FUNCTION_BLOCK ACVariobatch EXTENDS ACComponent IMPLEMENTS IACVariobatch
VAR_INPUT
END_VAR
VAR_OUTPUT
	// Metadata about Memory-Structure, Index in Array represents Instance-ID
	_Metadata : ARRAY [1..GCL.cMetaObjMAX] OF ACRMemoryMetaObj;
	// Copy of Memory
	_Memory : ARRAY [0..GCL.cMemorySizeMAX] OF BYTE;
	_MemorySizeUsed : UDINT;

	// Property-Changed-Notifications
	_EventsByte : ACRMemoryByteEvents;
	_EventsUInt : ACRMemoryUIntEvents;
	_EventsInt : ACRMemoryIntEvents;
	_EventsUDInt : ACRMemoryUDIntEvents;
	_EventsDInt : ACRMemoryDIntEvents;
	_EventsReal : ACRMemoryRealEvents;
	_EventsLReal : ACRMemoryLRealEvents;
	_EventsString : ACRMemoryStringEvents;
	_EventsTime : ACRMemoryTimeEvents;
	_EventsDT : ACRMemoryDTEvents;
	_EventCycleInfo : ACREventCycleInfo; 
	_MemPropEventCycle : ARRAY [1..GCL.cMetaObjMAX, 1..GCL.cMetaPropMAX] OF ACREventCycleProp;
	
	_InSimulation : BOOL;
	END_VAR
VAR
END_VAR

METHOD PUBLIC FB_postinit
VAR_INPUT
		root : IACVariobatch;
END_VAR
ResetMemory();
SUPER^.FB_postinit(root);
END_METHOD

PROPERTY InSimulation : BOOL
GET
InSimulation := _InSimulation;
END_GET
END_PROPERTY

METHOD OnObjectMetaBuilded
VAR_INPUT
	iObject : IACObject;
END_VAR
VAR
	instanceID : UDINT;
	memorySizeToObject : UDINT;
	i : UINT;
	offset : WORD;
END_VAR
instanceID := iObject.InstanceID;
offset := 0;

IF instanceID > 1 THEN
	_Metadata[instanceID]._OffsetInMemory := _Metadata[instanceID-1]._MetaPropSize + _Metadata[instanceID-1]._OffsetInMemory;
END_IF

IF iObject.MaxPropertyID >= 1 THEN
	FOR i:=1 TO iObject.MaxPropertyID BY 1
	  DO
		IF (_Metadata[instanceID]._MetaProp[i]._Length > 0) THEN
			_Metadata[instanceID]._MetaProp[i]._Offset := offset;
			offset := offset + _Metadata[instanceID]._MetaProp[i]._Length;
		//ELSE
			//EXIT;
		END_IF
	END_FOR;
END_IF

_Metadata[instanceID]._MaxPropertyID := iObject.MaxPropertyID;
_Metadata[instanceID]._MetaPropSize := offset;
memorySizeToObject := _Metadata[instanceID]._OffsetInMemory + offset;

IF _MemorySizeUsed < memorySizeToObject THEN
	_MemorySizeUsed := memorySizeToObject;
END_IF
END_METHOD

METHOD PUBLIC OnPropertyChangedBool
VAR_INPUT
	object : IACObject;
	propertyID : UINT;
	value : BOOL;
END_VAR
VAR
	instanceID : UDINT;
	memAdr : UDINT;
	eventIndex : DINT;
END_VAR
instanceID := object.InstanceID;
// 1. Copy to memory
memAdr := _Metadata[instanceID]._OffsetInMemory + _Metadata[instanceID]._MetaProp[propertyID]._Offset;
IF value THEN
	_Memory[memAdr] := 1;
ELSE
	_Memory[memAdr] := 0;
END_IF

// 2. Add to Eventlist
IF _EventCycleInfo._MemReadCycle = _EventCycleInfo._MemWriteCycle THEN
	IF _EventCycleInfo._MemWriteCycle > GCL.cMemoryEventCycleMAX THEN
		_EventCycleInfo._MemWriteCycle := 0;
	END_IF
	_EventCycleInfo._MemWriteCycle := _EventCycleInfo._MemWriteCycle + 1;
END_IF

IF _MemPropEventCycle[instanceID, propertyID]._MemWriteCycle = _EventCycleInfo._MemWriteCycle THEN
	eventIndex := _MemPropEventCycle[instanceID, propertyID]._MemEventPos;
ELSE
	eventIndex := _EventCycleInfo._NextByteEventIndex;
	IF eventIndex < 0 OR eventIndex > GCL.cMemoryEventsMAX THEN
		eventIndex := 0;
	END_IF	
	_MemPropEventCycle[instanceID, propertyID]._MemEventPos := eventIndex;
	_MemPropEventCycle[instanceID, propertyID]._MemWriteCycle := _EventCycleInfo._MemWriteCycle;
	_EventCycleInfo._NextByteEventIndex := eventIndex + 1;
END_IF

_EventsByte._Values[eventIndex]._InstanceID := instanceID;
_EventsByte._Values[eventIndex]._PropertyID := propertyID;
_EventsByte._Values[eventIndex]._Value := _Memory[memAdr];
END_METHOD

METHOD PUBLIC OnPropertyChangedByte
VAR_INPUT
	object : IACObject;
	propertyID : UINT;
	value : BYTE;
END_VAR
VAR
	instanceID : UDINT;
	memAdr : UDINT;
	eventIndex : DINT;
END_VAR
instanceID := object.InstanceID;

// 1. Copy to memory
memAdr := _Metadata[instanceID]._OffsetInMemory + _Metadata[instanceID]._MetaProp[propertyID]._Offset;
_Memory[memAdr] := value;

// 2. Add to Eventlist
IF _EventCycleInfo._MemReadCycle = _EventCycleInfo._MemWriteCycle THEN
	IF _EventCycleInfo._MemWriteCycle > GCL.cMemoryEventCycleMAX THEN
		_EventCycleInfo._MemWriteCycle := 0;
	END_IF
	_EventCycleInfo._MemWriteCycle := _EventCycleInfo._MemWriteCycle + 1;
END_IF

IF _MemPropEventCycle[instanceID, propertyID]._MemWriteCycle = _EventCycleInfo._MemWriteCycle THEN
	eventIndex := _MemPropEventCycle[instanceID, propertyID]._MemEventPos;
ELSE
	eventIndex := _EventCycleInfo._NextByteEventIndex;
	IF eventIndex < 0 OR eventIndex > GCL.cMemoryEventsMAX THEN
		eventIndex := 0;
	END_IF	
	_MemPropEventCycle[instanceID, propertyID]._MemEventPos := eventIndex;
	_MemPropEventCycle[instanceID, propertyID]._MemWriteCycle := _EventCycleInfo._MemWriteCycle;
	_EventCycleInfo._NextByteEventIndex := eventIndex + 1;
END_IF

_EventsByte._Values[eventIndex]._InstanceID := instanceID;
_EventsByte._Values[eventIndex]._PropertyID := propertyID;
_EventsByte._Values[eventIndex]._Value := value;
END_METHOD

METHOD PUBLIC OnPropertyChangedDInt
VAR_INPUT
	object : IACObject;
	propertyID : UINT;
	value : DINT;
END_VAR
VAR
	instanceID : UDINT;
	memAdr : UDINT;
	eventIndex : DINT;
END_VAR
instanceID := object.InstanceID;

// 1. Copy to memory
memAdr := _Metadata[instanceID]._OffsetInMemory + _Metadata[instanceID]._MetaProp[propertyID]._Offset;
MEMCPY(ADR(_Memory[memAdr]), ADR(value), GCL.cSizeDINT);

// 2. Add to Eventlist
IF _EventCycleInfo._MemReadCycle = _EventCycleInfo._MemWriteCycle THEN
	IF _EventCycleInfo._MemWriteCycle > GCL.cMemoryEventCycleMAX THEN
		_EventCycleInfo._MemWriteCycle := 0;
	END_IF
	_EventCycleInfo._MemWriteCycle := _EventCycleInfo._MemWriteCycle + 1;
END_IF

IF _MemPropEventCycle[instanceID, propertyID]._MemWriteCycle = _EventCycleInfo._MemWriteCycle THEN
	eventIndex := _MemPropEventCycle[instanceID, propertyID]._MemEventPos;
ELSE
	eventIndex := _EventCycleInfo._NextDIntEventIndex;
	IF eventIndex < 0 OR eventIndex > GCL.cMemoryEventsMAX THEN
		eventIndex := 0;
	END_IF	
	_MemPropEventCycle[instanceID, propertyID]._MemEventPos := eventIndex;
	_MemPropEventCycle[instanceID, propertyID]._MemWriteCycle := _EventCycleInfo._MemWriteCycle;
	_EventCycleInfo._NextDIntEventIndex := eventIndex + 1;
END_IF

_EventsDInt._Values[eventIndex]._InstanceID := instanceID;
_EventsDInt._Values[eventIndex]._PropertyID := propertyID;
_EventsDInt._Values[eventIndex]._Value := value;
END_METHOD

METHOD PUBLIC OnPropertyChangedDT
VAR_INPUT
	object : IACObject;
	propertyID : UINT;
	value : DATE_AND_TIME;
END_VAR
VAR
	instanceID : UDINT;
	memAdr : UDINT;
	eventIndex : DINT;
END_VAR
instanceID := object.InstanceID;

// 1. Copy to memory
memAdr := _Metadata[instanceID]._OffsetInMemory + _Metadata[instanceID]._MetaProp[propertyID]._Offset;
MEMCPY(ADR(_Memory[memAdr]), ADR(value), GCL.cSizeDT);

// 2. Add to Eventlist
IF _EventCycleInfo._MemReadCycle = _EventCycleInfo._MemWriteCycle THEN
	IF _EventCycleInfo._MemWriteCycle > GCL.cMemoryEventCycleMAX THEN
		_EventCycleInfo._MemWriteCycle := 0;
	END_IF
	_EventCycleInfo._MemWriteCycle := _EventCycleInfo._MemWriteCycle + 1;
END_IF

IF _MemPropEventCycle[instanceID, propertyID]._MemWriteCycle = _EventCycleInfo._MemWriteCycle THEN
	eventIndex := _MemPropEventCycle[instanceID, propertyID]._MemEventPos;
ELSE
	eventIndex := _EventCycleInfo._NextDTEventIndex;
	IF eventIndex < 0 OR eventIndex > GCL.cMemoryEventsMidMAX THEN
		eventIndex := 0;
	END_IF	
	_MemPropEventCycle[instanceID, propertyID]._MemEventPos := eventIndex;
	_MemPropEventCycle[instanceID, propertyID]._MemWriteCycle := _EventCycleInfo._MemWriteCycle;
	_EventCycleInfo._NextDTEventIndex := eventIndex + 1;
END_IF

_EventsDT._Values[eventIndex]._InstanceID := instanceID;
_EventsDT._Values[eventIndex]._PropertyID := propertyID;
_EventsDT._Values[eventIndex]._Value := value;
END_METHOD

METHOD PUBLIC OnPropertyChangedInt
VAR_INPUT
	object : IACObject;
	propertyID : UINT;
	value : INT;
END_VAR
VAR
	instanceID : UDINT;
	memAdr : UDINT;
	eventIndex : DINT;
END_VAR
instanceID := object.InstanceID;

// 1. Copy to memory
memAdr := _Metadata[instanceID]._OffsetInMemory + _Metadata[instanceID]._MetaProp[propertyID]._Offset;
MEMCPY(ADR(_Memory[memAdr]), ADR(value), GCL.cSizeINT);

// 2. Add to Eventlist
IF _EventCycleInfo._MemReadCycle = _EventCycleInfo._MemWriteCycle THEN
	IF _EventCycleInfo._MemWriteCycle > GCL.cMemoryEventCycleMAX THEN
		_EventCycleInfo._MemWriteCycle := 0;
	END_IF
	_EventCycleInfo._MemWriteCycle := _EventCycleInfo._MemWriteCycle + 1;
END_IF

IF _MemPropEventCycle[instanceID, propertyID]._MemWriteCycle = _EventCycleInfo._MemWriteCycle THEN
	eventIndex := _MemPropEventCycle[instanceID, propertyID]._MemEventPos;
ELSE
	eventIndex := _EventCycleInfo._NextIntEventIndex;
	IF eventIndex < 0 OR eventIndex > GCL.cMemoryEventsMAX THEN
		eventIndex := 0;
	END_IF	
	_MemPropEventCycle[instanceID, propertyID]._MemEventPos := eventIndex;
	_MemPropEventCycle[instanceID, propertyID]._MemWriteCycle := _EventCycleInfo._MemWriteCycle;
	_EventCycleInfo._NextIntEventIndex := eventIndex + 1;
END_IF

_EventsInt._Values[eventIndex]._InstanceID := instanceID;
_EventsInt._Values[eventIndex]._PropertyID := propertyID;
_EventsInt._Values[eventIndex]._Value := value;
END_METHOD

METHOD PUBLIC OnPropertyChangedLReal
VAR_INPUT
	object : IACObject;
	propertyID : UINT;
	value : LREAL;
END_VAR
VAR
	instanceID : UDINT;
	memAdr : UDINT;
	eventIndex : DINT;
END_VAR
instanceID := object.InstanceID;

// 1. Copy to memory
memAdr := _Metadata[instanceID]._OffsetInMemory + _Metadata[instanceID]._MetaProp[propertyID]._Offset;
MEMCPY(ADR(_Memory[memAdr]), ADR(value), GCL.cSizeLREAL);

// 2. Add to Eventlist
IF _EventCycleInfo._MemReadCycle = _EventCycleInfo._MemWriteCycle THEN
	IF _EventCycleInfo._MemWriteCycle > GCL.cMemoryEventCycleMAX THEN
		_EventCycleInfo._MemWriteCycle := 0;
	END_IF
	_EventCycleInfo._MemWriteCycle := _EventCycleInfo._MemWriteCycle + 1;
END_IF

IF _MemPropEventCycle[instanceID, propertyID]._MemWriteCycle = _EventCycleInfo._MemWriteCycle THEN
	eventIndex := _MemPropEventCycle[instanceID, propertyID]._MemEventPos;
ELSE
	eventIndex := _EventCycleInfo._NextLRealEventIndex;
	IF eventIndex < 0 OR eventIndex > GCL.cMemoryEventsMAX THEN
		eventIndex := 0;
	END_IF	
	_MemPropEventCycle[instanceID, propertyID]._MemEventPos := eventIndex;
	_MemPropEventCycle[instanceID, propertyID]._MemWriteCycle := _EventCycleInfo._MemWriteCycle;
	_EventCycleInfo._NextLRealEventIndex := eventIndex + 1;
END_IF

_EventsLReal._Values[eventIndex]._InstanceID := instanceID;
_EventsLReal._Values[eventIndex]._PropertyID := propertyID;
_EventsLReal._Values[eventIndex]._Value := value;
END_METHOD

METHOD PUBLIC OnPropertyChangedReal
VAR_INPUT
	object : IACObject;
	propertyID : UINT;
	value : REAL;
END_VAR
VAR
	instanceID : UDINT;
	memAdr : UDINT;
	eventIndex : DINT;
END_VAR
instanceID := object.InstanceID;

// 1. Copy to memory
memAdr := _Metadata[instanceID]._OffsetInMemory + _Metadata[instanceID]._MetaProp[propertyID]._Offset;
MEMCPY(ADR(_Memory[memAdr]), ADR(value), GCL.cSizeREAL);

// 2. Add to Eventlist
IF _EventCycleInfo._MemReadCycle = _EventCycleInfo._MemWriteCycle THEN
	IF _EventCycleInfo._MemWriteCycle > GCL.cMemoryEventCycleMAX THEN
		_EventCycleInfo._MemWriteCycle := 0;
	END_IF
	_EventCycleInfo._MemWriteCycle := _EventCycleInfo._MemWriteCycle + 1;
END_IF

IF _MemPropEventCycle[instanceID, propertyID]._MemWriteCycle = _EventCycleInfo._MemWriteCycle THEN
	eventIndex := _MemPropEventCycle[instanceID, propertyID]._MemEventPos;
ELSE
	eventIndex := _EventCycleInfo._NextRealEventIndex;
	IF eventIndex < 0 OR eventIndex > GCL.cMemoryEventsMAX THEN
		eventIndex := 0;
	END_IF	
	_MemPropEventCycle[instanceID, propertyID]._MemEventPos := eventIndex;
	_MemPropEventCycle[instanceID, propertyID]._MemWriteCycle := _EventCycleInfo._MemWriteCycle;
	_EventCycleInfo._NextRealEventIndex := eventIndex + 1;
END_IF

_EventsReal._Values[eventIndex]._InstanceID := instanceID;
_EventsReal._Values[eventIndex]._PropertyID := propertyID;
_EventsReal._Values[eventIndex]._Value := value;
END_METHOD

METHOD PUBLIC OnPropertyChangedString
VAR_INPUT
	object : IACObject;
	propertyID : UINT;
	value : STRING(255);
END_VAR
VAR
	instanceID : UDINT;
	memAdr : UDINT;
	eventIndex : DINT;
END_VAR
instanceID := object.InstanceID;

// 1. Copy to memory
memAdr := _Metadata[instanceID]._OffsetInMemory + _Metadata[instanceID]._MetaProp[propertyID]._Offset;
MEMCPY(ADR(_Memory[memAdr]), ADR(value), GCL.cSizeINT);

// 2. Add to Eventlist
IF _EventCycleInfo._MemReadCycle = _EventCycleInfo._MemWriteCycle THEN
	IF _EventCycleInfo._MemWriteCycle > GCL.cMemoryEventCycleMAX THEN
		_EventCycleInfo._MemWriteCycle := 0;
	END_IF
	_EventCycleInfo._MemWriteCycle := _EventCycleInfo._MemWriteCycle + 1;
END_IF

IF _MemPropEventCycle[instanceID, propertyID]._MemWriteCycle = _EventCycleInfo._MemWriteCycle THEN
	eventIndex := _MemPropEventCycle[instanceID, propertyID]._MemEventPos;
ELSE
	eventIndex := _EventCycleInfo._NextStringEventIndex;
	IF eventIndex < 0 OR eventIndex > GCL.cMemoryEventsSmallMAX THEN
		eventIndex := 0;
	END_IF	
	_MemPropEventCycle[instanceID, propertyID]._MemEventPos := eventIndex;
	_MemPropEventCycle[instanceID, propertyID]._MemWriteCycle := _EventCycleInfo._MemWriteCycle;
	_EventCycleInfo._NextStringEventIndex := eventIndex + 1;
END_IF

_EventsString._Values[eventIndex]._InstanceID := instanceID;
_EventsString._Values[eventIndex]._PropertyID := propertyID;
_EventsString._Values[eventIndex]._Value := value;
END_METHOD

METHOD OnPropertyChangedTime
VAR_INPUT
	object : IACObject;
	propertyID : UINT;
	value : TIME;
END_VAR
VAR
	instanceID : UDINT;
	memAdr : UDINT;
	eventIndex : DINT;
END_VAR
instanceID := object.InstanceID;

// 1. Copy to memory
memAdr := _Metadata[instanceID]._OffsetInMemory + _Metadata[instanceID]._MetaProp[propertyID]._Offset;
MEMCPY(ADR(_Memory[memAdr]), ADR(value), GCL.cSizeTIME);

// 2. Add to Eventlist
IF _EventCycleInfo._MemReadCycle = _EventCycleInfo._MemWriteCycle THEN
	IF _EventCycleInfo._MemWriteCycle > GCL.cMemoryEventCycleMAX THEN
		_EventCycleInfo._MemWriteCycle := 0;
	END_IF
	_EventCycleInfo._MemWriteCycle := _EventCycleInfo._MemWriteCycle + 1;
END_IF

IF _MemPropEventCycle[instanceID, propertyID]._MemWriteCycle = _EventCycleInfo._MemWriteCycle THEN
	eventIndex := _MemPropEventCycle[instanceID, propertyID]._MemEventPos;
ELSE
	eventIndex := _EventCycleInfo._NextTimeEventIndex;
	IF eventIndex < 0 OR eventIndex > GCL.cMemoryEventsMidMAX THEN
		eventIndex := 0;
	END_IF	
	_MemPropEventCycle[instanceID, propertyID]._MemEventPos := eventIndex;
	_MemPropEventCycle[instanceID, propertyID]._MemWriteCycle := _EventCycleInfo._MemWriteCycle;
	_EventCycleInfo._NextTimeEventIndex := eventIndex + 1;
END_IF

_EventsTime._Values[eventIndex]._InstanceID := instanceID;
_EventsTime._Values[eventIndex]._PropertyID := propertyID;
_EventsTime._Values[eventIndex]._Value := value;
END_METHOD

METHOD PUBLIC OnPropertyChangedUDInt
VAR_INPUT
	object : IACObject;
	propertyID : UINT;
	value : UDINT;
END_VAR
VAR
	instanceID : UDINT;
	memAdr : UDINT;
	eventIndex : DINT;
END_VAR
instanceID := object.InstanceID;

// 1. Copy to memory
memAdr := _Metadata[instanceID]._OffsetInMemory + _Metadata[instanceID]._MetaProp[propertyID]._Offset;
MEMCPY(ADR(_Memory[memAdr]), ADR(value), GCL.cSizeUDINT);

// 2. Add to Eventlist
IF _EventCycleInfo._MemReadCycle = _EventCycleInfo._MemWriteCycle THEN
	IF _EventCycleInfo._MemWriteCycle > GCL.cMemoryEventCycleMAX THEN
		_EventCycleInfo._MemWriteCycle := 0;
	END_IF
	_EventCycleInfo._MemWriteCycle := _EventCycleInfo._MemWriteCycle + 1;
END_IF

IF _MemPropEventCycle[instanceID, propertyID]._MemWriteCycle = _EventCycleInfo._MemWriteCycle THEN
	eventIndex := _MemPropEventCycle[instanceID, propertyID]._MemEventPos;
ELSE
	eventIndex := _EventCycleInfo._NextUDintEventIndex;
	IF eventIndex < 0 OR eventIndex > GCL.cMemoryEventsMAX THEN
		eventIndex := 0;
	END_IF	
	_MemPropEventCycle[instanceID, propertyID]._MemEventPos := eventIndex;
	_MemPropEventCycle[instanceID, propertyID]._MemWriteCycle := _EventCycleInfo._MemWriteCycle;
	_EventCycleInfo._NextUDintEventIndex := eventIndex + 1;
END_IF

_EventsUDInt._Values[eventIndex]._InstanceID := instanceID;
_EventsUDInt._Values[eventIndex]._PropertyID := propertyID;
_EventsUDInt._Values[eventIndex]._Value := value;
END_METHOD

METHOD PUBLIC OnPropertyChangedUInt
VAR_INPUT
	object : IACObject;
	propertyID : UINT;
	value : UINT;
END_VAR
VAR
	instanceID : UDINT;
	memAdr : UDINT;
	eventIndex : DINT;
END_VAR
instanceID := object.InstanceID;

// 1. Copy to memory
memAdr := _Metadata[instanceID]._OffsetInMemory + _Metadata[instanceID]._MetaProp[propertyID]._Offset;
MEMCPY(ADR(_Memory[memAdr]), ADR(value), GCL.cSizeUINT);

// 2. Add to Eventlist
IF _EventCycleInfo._MemReadCycle = _EventCycleInfo._MemWriteCycle THEN
	IF _EventCycleInfo._MemWriteCycle > GCL.cMemoryEventCycleMAX THEN
		_EventCycleInfo._MemWriteCycle := 0;
	END_IF
	_EventCycleInfo._MemWriteCycle := _EventCycleInfo._MemWriteCycle + 1;
END_IF

IF _MemPropEventCycle[instanceID, propertyID]._MemWriteCycle = _EventCycleInfo._MemWriteCycle THEN
	eventIndex := _MemPropEventCycle[instanceID, propertyID]._MemEventPos;
ELSE
	eventIndex := _EventCycleInfo._NextUIntEventIndex;
	IF eventIndex < 0 OR eventIndex > GCL.cMemoryEventsMAX THEN
		eventIndex := 0;
	END_IF	
	_MemPropEventCycle[instanceID, propertyID]._MemEventPos := eventIndex;
	_MemPropEventCycle[instanceID, propertyID]._MemWriteCycle := _EventCycleInfo._MemWriteCycle;
	_EventCycleInfo._NextUIntEventIndex := eventIndex + 1;
END_IF

_EventsUInt._Values[eventIndex]._InstanceID := instanceID;
_EventsUInt._Values[eventIndex]._PropertyID := propertyID;
_EventsUInt._Values[eventIndex]._Value := value;
END_METHOD

METHOD PROTECTED ResetMemory
VAR_INPUT
END_VAR
//MEMSET(ADR(_Memory), 0, GCL.cMemorySizeMAX+1);
MEMSET(ADR(_Memory), 0, SIZEOF(_Memory));
MEMSET(ADR(_Metadata), 0, SIZEOF(_Metadata));
MEMSET(ADR(_MemPropEventCycle), 0, SIZEOF(_MemPropEventCycle));
_EventCycleInfo._NextByteEventIndex := -1;
_EventCycleInfo._NextUIntEventIndex := -1;
_EventCycleInfo._NextIntEventIndex := -1;
_EventCycleInfo._NextUDIntEventIndex := -1;
_EventCycleInfo._NextDIntEventIndex := -1;
_EventCycleInfo._NextRealEventIndex := -1;
_EventCycleInfo._NextLRealEventIndex := -1;
_EventCycleInfo._NextStringEventIndex := -1;
_EventCycleInfo._NextTimeEventIndex := -1;
_EventCycleInfo._NextDTEventIndex := -1;
_EventCycleInfo._MemReadCycle := 0;
_EventCycleInfo._MemWriteCycle := 0;
END_METHOD

METHOD SetCompMetadata
VAR_INPUT
	iObject : IACObject;
END_VAR
_Metadata[iObject.InstanceID]._ACUrl := iObject.ACUrlS;
_Metadata[iObject.InstanceID]._TypeOfACObject := iObject.TypeofACObject;
END_METHOD

METHOD SetPropMetadata
VAR_INPUT
	iObject : IACObject;
	propertyID : UINT;
	sizeOfPropType : UINT;
END_VAR
VAR
	instanceID : UDINT;
END_VAR
instanceID := iObject.InstanceID;
_Metadata[instanceID]._MetaProp[propertyID]._Length := sizeOfPropType;
//_Metadata[iObject.InstanceID]._MetaProp[propertyID]._Length := sizeOfPropType;
END_METHOD

END_FUNCTION_BLOCK

(* stored: Version 1.1.0.1, ProductVersion 3.1.4022.7
   POU ACVariobatch: Id {7f8371af-ea2e-4d7b-b646-a4060fb5ca8e}, SpecialFunc None
   Method FB_postinit: Id {a5b017b7-3729-4798-ad4b-68e0e9ad0b9c}
   Property InSimulation: Id {193e4ead-fa0f-4c63-9189-3ffaf504a0ef}
   Get Get: Id {fd5609e9-c948-40bc-8cc0-adcfaea76a01}
   Method OnObjectMetaBuilded: Id {699a95d3-ba50-4fcc-8b80-9f9023265d60}
   Method OnPropertyChangedBool: Id {20747f1d-e5ae-4f9c-87ef-66214f330c31}
   Method OnPropertyChangedByte: Id {7c9b4f3c-326b-467a-9381-eeef07921337}
   Method OnPropertyChangedDInt: Id {c0c87217-11d2-4fd9-8b72-07d6398d67a3}
   Method OnPropertyChangedDT: Id {7f04dc80-8108-42a0-8cc6-825c9fb51a99}
   Method OnPropertyChangedInt: Id {d2794bf4-c324-4e3b-a381-63ecad48aa08}
   Method OnPropertyChangedLReal: Id {e3eafae1-71ce-4881-8862-ce3909504fd0}
   Method OnPropertyChangedReal: Id {2ca7d0af-3283-4c26-a6db-d965870c9e74}
   Method OnPropertyChangedString: Id {87de1059-8957-4e97-b6a7-ed8c77a3958c}
   Method OnPropertyChangedTime: Id {8a83e0b6-c18c-4fd5-94f3-ee8ad0737790}
   Method OnPropertyChangedUDInt: Id {773dab02-abd4-4720-9ce8-4285dc5ce1d5}
   Method OnPropertyChangedUInt: Id {66833e0c-c2b0-48ed-b372-794b0a3cc0fe}
   Method ResetMemory: Id {18add70c-5930-45a2-929c-a87e5cd576c3}
   Method SetCompMetadata: Id {a9cb9b8f-e1d5-466a-a3c1-79b3c5fe1bf3}
   Method SetPropMetadata: Id {fa04dda8-bb96-4132-b850-f807b2b90a29} *)
